// A move profile only provide velocity and its derivatives
TYPE MoveProfile_t :
STRUCT
    lrVelocity  : LREAL;         // Velocity to position
    lrAccel     : LREAL;         // acceleration to position
    lrDecel     : LREAL;         // deceleration to position
    lrJerk      : LREAL;         // jerk to position
END_STRUCT
END_TYPE

(* stored: Version 1.1.0.1, ProductVersion 3.1.4024.6
   DUT MoveProfile_t: Id {ce3ac506-cbab-4386-bc87-7e0bc71eb7f0} *)
